{attribute 'hide_all_locals'}
{attribute 'enable_dynamic_creation'}
FUNCTION_BLOCK FB_ShapeCreator  EXTENDS FB_AbstractFactory
VAR_INPUT
END_VAR
VAR_OUTPUT
END_VAR
VAR
      pCircle    : POINTER TO FB_Circle;
      pRectangle : POINTER TO FB_Rectangle;
      pSquare    : POINTER TO FB_Square;
      pStar      : POINTER TO FB_Star;
      pTriangle  : POINTER TO FB_Triangle;
      iShape 	 : I_Shape;
END_VAR

METHOD FB_exit : BOOL
VAR_INPUT
	bInCopyCode : BOOL; // if TRUE, the exit method is called for exiting an instance that is copied afterwards (online change).
END_VAR
IF (pCircle <> 0) THEN
  __DELETE(pCircle);
  pCircle := 0;
END_IF

IF (pRectangle <> 0) THEN
  __DELETE(pRectangle);
  pRectangle := 0;
END_IF

IF (pSquare <> 0) THEN
  __DELETE(pSquare);
  pSquare := 0;
END_IF

IF (pStar <> 0) THEN
  __DELETE(pStar);
  pStar := 0;
END_IF

IF (pTriangle <> 0) THEN
  __DELETE(pTriangle);
  pTriangle := 0;
END_IF
END_METHOD

METHOD M_GetShapeObject : I_shape
VAR_INPUT
	eShape : E_Shape;
END_VAR
CASE eShape OF
	E_Shape.Circle:
		
		//Dynamic instantiation  
		pCircle := __NEW(FB_Circle);
		iShape := pCircle^;
		
		//Return the object
		IF iShape <> 0 THEN
			M_GetShapeObject := iShape;
		END_IF
		
		//Release the memory
		IF (pCircle <> 0) THEN
			__DELETE(pCircle);
			pCircle := 0;
		END_IF
		
		eShape := E_Shape.init;
	
	E_Shape.Rectangle:
		pRectangle := __NEW(FB_Rectangle);
		iShape := pRectangle^;
		
		//Return the object
		IF iShape <> 0 THEN
			M_GetShapeObject := iShape;
		END_IF
		
		IF (pRectangle <> 0) THEN
			__DELETE(pRectangle);
			pRectangle := 0;
		END_IF
		
		eShape := E_Shape.init;	
		
	E_Shape.Sqaure:
		pSquare := __NEW(FB_Square);
		iShape := pSquare^;
		
		//Return the object
		IF iShape <> 0 THEN
			M_GetShapeObject := iShape;
		END_IF
		
		IF (pSquare <> 0) THEN
			__DELETE(pSquare);
			pSquare := 0;
		END_IF
		
		eShape := E_Shape.init;	

	E_Shape.Star:
		pStar := __NEW(FB_Star);
		iShape := pStar^;
		
		//Return the object
		IF iShape <> 0 THEN
			M_GetShapeObject := iShape;
		END_IF
		
		IF (pStar <> 0) THEN
			__DELETE(pStar);
			pStar := 0;
		END_IF
		
		eShape := E_Shape.init;	
	
	E_Shape.Triangle:
		pTriangle := __NEW(FB_Triangle);
		iShape := pTriangle^;
		
		//Return the object
		IF iShape <> 0 THEN
			M_GetShapeObject := iShape;
		END_IF
		
		IF (pTriangle <> 0) THEN
			__DELETE(pTriangle);
			pTriangle := 0;
		END_IF
		
		eShape := E_Shape.init;	
END_CASE
END_METHOD

METHOD M_ReleaseMemory : BOOL
VAR_INPUT
END_VAR
IF (pCircle <> 0) THEN
  __DELETE(pCircle);
  pCircle := 0;
END_IF

IF (pRectangle <> 0) THEN
  __DELETE(pRectangle);
  pRectangle := 0;
END_IF

IF (pSquare <> 0) THEN
  __DELETE(pSquare);
  pSquare := 0;
END_IF

IF (pStar <> 0) THEN
  __DELETE(pStar);
  pStar := 0;
END_IF

IF (pTriangle <> 0) THEN
  __DELETE(pTriangle);
  pTriangle := 0;
END_IF
END_METHOD

END_FUNCTION_BLOCK

(* stored: Version 1.1.0.1, ProductVersion 3.1.4024.12
   POU FB_ShapeCreator: Id {54fca42c-4fe0-4907-9486-763b9701f91b}, SpecialFunc None
   Method FB_exit: Id {cb977582-9888-4ce3-981b-67b2b727f525}
   Method M_GetShapeObject: Id {be126036-b314-4968-ac3b-33ff3962266f}
   Method M_ReleaseMemory: Id {6e326109-079b-4b95-9c22-3c9f3b81cb07} *)
